// TIA Portal V20 export
TYPE "LER_typeAlignMoveCalibrationInterface"
// stored: Access Published
   STRUCT
      commands : "LER_typeAlignMoveCalibrationCommands";
      monitoring : "LER_typeAlignMoveCalibrationMonitoring";
      configuration : "LER_typeAlignMoveCalibrationConfiguration";
   END_STRUCT;
END_TYPE
